# B&R Automation Studio project MIG1 (part 6)

```c
					ax = 0;
					for(k = 0 ; k < mgr->hrdw[i].AxisNum ; k++){

						if(mgr->pAxis[i]){
							if((mgr->pAxis[i][k].AxisID & 0x00FF)== SenderID){
								ax = &mgr->pAxis[i][k];
								break;

							}
						}

					}
					if(!ax)
						return 0;

#ifdef KK_SUPER_TRACE
					KK_Ind_RcvMsg_Cntr[i][k]++;
#endif
					/////////////////////////////////////////////////////////////
					// Parse message //
					// Firmware version
					if((*pRxCANidentifier) == 0xD80A0009){

						mgr->Firmware[i] = ((UDINT)pRxCANdata[1] + ((UDINT)pRxCANdata[0] <<16));
					}

					///////////////////////////////////////////////////////
					/*Received 32-bit variable*/
					else if((*pRxCANidentifier)& 0x800){ /* Check if 16 or 32-bit variable - bit 11 */

						if(pRxCANdata[0] == 0x090E){ /* Status Received */

							ax->Flag |= 0x0C; //bit 2 & 3  (* New Status received *)
							ax->DriveStatusRegisterL = pRxCANdata[1];
							ax->DriveStatusRegisterH = pRxCANdata[2];

						}
						else{ /* General variable received. Save address to Axis structure*/
							ax->Flag |= 0x01; //bit 0 (* New Variable received *)

							ax->VarAddress = pRxCANdata[0];
							ax->DataLow  = pRxCANdata[1];
							ax->DataHigh = pRxCANdata[2];

						}
					}
					////////////////////////////////////////////
					/*Received 16-bit variable*/
					else if(pRxCANdata[0] == 0x08FC){  /* MER register received */
						if(pRxCANdata[1] && 0xFFEF){ // Mask Serial comunnication error
							ax->Flag |= 0x02; //bit 1 (* New Error received *)
							ax->DriveErrorRegister = pRxCANdata[1];
						}
					}
					/***********/
					else if(pRxCANdata[0] == 0x0863){  /* PVT status register received*/

						ax->Flag |= 0x10; //bit 4 (* New PVT status received *)
						ax->PVTstatus = pRxCANdata[1];

					}
					/***********/
					else {  /* other variable received*/

						ax->Flag |= 0x01; //bit 0 (* New Variable received *)
						ax->VarAddress = pRxCANdata[0];
						ax->DataLow  = pRxCANdata[1];

					}

			}

		}
	}

return 1;
}

DINT ReadValue(char **p, DINT *val){

	if(*p == strchr(*p , 0x0D)){
		(*p)+= 2;
		return -1;
	}

	else {

		*val = 0;

		while( (**p != 0x0D) || (**p != 0x0A)){

			if((**p >= '0') && (**p <= '9')){
				*val = *val<<4;
				*val += (**p) - '0';
			}
			else if((**p >= 'A') && (**p <= 'F')){
				*val = *val<<4;
				*val += (**p) - 'A' + 10;
			}
			else{
				(*p)++;
				break;
			}

			(*p)++;

		}

	}

	(*p)++;

return 1;
}

DINT CalcUnits(TML_typ* tml){

	if( (tml->_cfg.rev_motor != 0.0) && (tml->_cfg.loopPeriod > 0)){
		tml->_int.kPos = (tml->_cfg.units * fabsf(tml->_cfg.rev_motor)) * tml->_cfg.rev_scale ;
		tml->_int.kVel = fabsf(tml->_int.kPos * tml->_cfg.loopPeriod);
		tml->_int.kAcc = tml->_int.kVel * tml->_cfg.loopPeriod ;
		//tml->_int.PVTPeriod = 0.02/ tml->_cfg.loopPeriod;
		tml->_int.PVTPeriod = (UINT)(tml->_cfg.PVTPeriod / tml->_cfg.loopPeriod + 0.5);
		return 1;
	}
	else
		return -1;

return 1;
}

DINT TML_InterpretMessage_UDP(TML_MGR_typ* mgr){

USINT *pCountRegister;
UDINT *pRxCANidentifier ;
UINT *pRxCANdata;
TML_Axis_typ *ax;
RS_Channel_typ *data , *data_sent;
USINT SenderID;
UINT i , k , n;
plcstring _str[128];
UINT adr ;
//UDINT val , *pVal;
USINT dataType; // 0 - no data , 1 - 16 data , 2 - 32 data
UINT *pUINT , val_UINT[2];

	if(!mgr)
		return -1;

	//pVal = &val;
	pUINT = &val_UINT[0];

	for(n = 0 ; n < 2 ; n++){ // Two channels

		data = ((RS_Channel_typ*)mgr->pRecData[n]) ;

		data_sent = ((RS_Channel_typ*)mgr->pSendData[n]) ;

		if(!data || !data_sent)
			continue;

		////////////////////////////////////////////////////////////////
		//////   New from 6 June 2023

		if(data->Len == 0)
			continue;

		mgr->hrdw[n].RXCount++;

		//if((data_sent->Len == 0)
		if(data->Len == 1){

			if(data->Data[0] == 0x4F){
				//&& (data_sent->Status == 0x1)){

				//LogTxt(&LogMgr, "ACK: F%d T%d" , (UDINT)mgr->hrdw[n].TXCountReadBack , (UDINT)mgr->hrdw[n].TXCount);
				data->Msg_ID ++;
				if(data_sent->Msg_ID == data->Msg_ID){

					mgr->hrdw[n].TXCountReadBack = mgr->hrdw[n].TXCount;
					data->Msg_ID = data_sent->Msg_ID;
					data->Status++;

				}else{

					mgr->hrdw[n].TXCountReadBack = mgr->hrdw[n].TXCount;
					data->Msg_ID = data_sent->Msg_ID;
					data_sent->Msg_Error++;
					data->Msg_Error++;
				}

			}
			else {
				data_sent->Trash_Cntr++;
				data->Trash_Cntr++;
			}

			data->Len = 0;
			continue;
		}

		//StreamToHex(data->Data, _str, data->Len);
		//LogTxt(&LogMgr, "%d-%d R: %s" , (UDINT) n , data->Len, _str);

		if(((data->Len != 10) && (data->Len != 12)&&(data->Len != 14) )){ // 16 or 32 bit TakeData only
			data->Trash_Cntr++;
			data->Len = 0;
			continue;

		}

		//if(!(data->Data[1] == 0x00 && data->Data[2] == 0xA1)){ // Not for me
		if(!((data->Data[1] == 0x00) && (data->Data[2] == (HOST_ID*0x10 +1)))){ // Not for me
			data->Trash_Cntr++;
			data->Len = 0;
			continue;
		}

		///////////////////////////////////////////////////////////////
		///////////////////////////////////////////////////////////////

		/*
		if((data_sent->Len == 0)
			&& (data->Len == 1)
			&& (data->Data[0] == 0x4F)){
			//&& (data_sent->Status == 0x1)){

			//LogTxt(&LogMgr, "ACK: F%d T%d" , (UDINT)mgr->hrdw[n].TXCountReadBack , (UDINT)mgr->hrdw[n].TXCount);

			mgr->hrdw[n].TXCountReadBack = mgr->hrdw[n].TXCount;

			data->Status++;

		}

		if(data->Len == 0)
			continue;

		//StreamToHex(data->Data, _str, data->Len);
		//LogTxt(&LogMgr, "%d-%d R: %s" , (UDINT) n , data->Len, _str);

		mgr->hrdw[n].RXCount++;

		if((data->Len == 1) // 0x4F - confirmation of cmd
			||((data->Len != 10) && (data->Len != 12)&&(data->Len != 14) )){ // 16 or 32 bit TakeData only

			data->Len = 0;
			return 0;

		}

		//if(!(data->Data[1] == 0x00 && data->Data[2] == 0xA1)){ // Not for me
		if(!((data->Data[1] == 0x00) && (data->Data[2] == (HOST_ID*0x10 +1)))){ // Not for me
			data->Len = 0;
			return;
		}

		*/
		///////////////// to dziala ///////////////////////
		dataType = 0;
		//val = 0;
		val_UINT[0] = 0;
		val_UINT[1] = 0;
		switch(data->Data[3]){

			case 0xB4: // TakeData 16 bit 0r 32 bit

				SenderID = (UINT)data->Data[6] + (UINT)data->Data[5] * 0x100;
				SenderID /= 0x10;

				adr = (UINT)data->Data[8] + (UINT)data->Data[7] * 0x100;

				switch(data->Data[4]){

					case 0x04: // 16 bit data

						*((char*)pUINT) = data->Data[10];
						*((char*)pUINT + 1) = data->Data[9];

						dataType = 1;

					break;

					case 0x05: // 32 bit data

						//val = (UINT)data->Data[10] + (UINT)data->Data[9] * 0x100 \
							//+ (UINT)data->Data[12] * 0x10000  + (UINT)data->Data[11] * 0x1000000;

						//*((char*)pVal) = data->Data[10];
						//*((char*)pVal + 1) = data->Data[9];
						//*((char*)pVal + 2) = data->Data[12];
						//*((char*)pVal + 3) = data->Data[11];

						*((char*)pUINT) = data->Data[10];
						*((char*)pUINT + 1) = data->Data[9];
						*((char*)pUINT + 2) = data->Data[12];
						*((char*)pUINT + 3) = data->Data[11];

						dataType = 2;

					break;

					default:

					break;
				}

				//LogTxt(&LogMgr, "D1:%d A:%X U: %X , %X" , (DINT)SenderID , (UINT)adr , val_UINT[0] , val_UINT[1]);

			break;

			case 0xD4: // TakeData2 16 bit
			case 0xD5: // TakeData2 32 bit

				SenderID = data->Data[4];

				adr = (UINT)data->Data[6] + (UINT)data->Data[5] * 0x100;

				switch(data->Data[3]){

					case 0xD4: // TakeData2 16 bit

						*((char*)pUINT) = data->Data[8];
						*((char*)pUINT + 1) = data->Data[7];

						dataType = 1;

					break;

					case 0xD5: // TakeData2 32 bit

						*((char*)pUINT) = data->Data[8];
						*((char*)pUINT + 1) = data->Data[7];
						*((char*)pUINT + 2) = data->Data[10];
						*((char*)pUINT + 3) = data->Data[9];

						dataType = 2;

					break;

				}

				//LogTxt(&LogMgr, "D2:%d A:%X U: %X , %X" , (DINT)SenderID , (UINT)adr  , val_UINT[0] , val_UINT[1]);

			break;

		}

		data->Len = 0;

		///////////////////////////////////////////////////////////////////////////
		ax = 0;
		for(k = 0 ; k < mgr->hrdw[n].AxisNum ; k++){

			if(mgr->pAxis[n]){
				if((mgr->pAxis[n][k].AxisID & 0x00FF)== SenderID){
					ax = &mgr->pAxis[n][k];
					//LogTxt(&LogMgr, "Axis Chan: %d Item: %d Node:%d Type: %d" , (UDINT) n , (UDINT)k , (UDINT)SenderID , (UDINT)dataType);
					break;

				}
			}

		}

		if(!ax)
			return 0;

		//ax->VarAddress = dataType;
		//ax->PVTstatus = SenderID;
		//return;

		//LogTxt(&LogMgr, "Type: %d Adr: %X U1:%X U2: %X " ,(UDINT)dataType , (UDINT)adr , (UDINT)val_UINT[0] , (UDINT)val_UINT[1] );

		switch(dataType){

			case 0: // nothing

			break;

			case 1: // 16 bit

				if(adr == 0x08FC){  /* MER register received */

					ax->AxisState = val_UINT[0] & 0xA000 ; // only enable and undervoltage

					if(val_UINT[0] & 0xFFEF){ // Mask Serial comunnication error
					//if(val_UINT[0] & 0x5FEF){ // Mask Serial comunnication error and  enable and undervoltage
						ax->Flag |= 0x02; //bit 1 (* New Error received *)
						ax->DriveErrorRegister = val_UINT[0];
					}
				}
				/***********/
				else if(adr == 0x0863){  /* PVT status register received*/

					ax->Flag |= 0x10; //bit 4 (* New PVT status received *)
					ax->PVTstatus = val_UINT[0];

				}
				/***********/
				else {	/* other variable received*/

					ax->Flag |= 0x01; //bit 0 (* New Variable received *)
					ax->VarAddress = adr;
					ax->DataLow  = val_UINT[0];

				}
			break;

			case 2: // 32 bit

				if(adr == 0x090E){ // Status Received

					ax->Flag |= 0x0C; //bit 2 & 3  New Status received
					ax->DriveStatusRegisterL = val_UINT[0];
					ax->DriveStatusRegisterH = val_UINT[1];

				}
				else{ // General variable received. Save address to Axis structure
					ax->Flag |= 0x01; //bit 0  New Variable received

					ax->VarAddress = adr;
					ax->DataLow  = val_UINT[0];
					ax->DataHigh = val_UINT[1];

				}

			break;

		}

		///////////////////////////////

	}

return 1;

}

DINT TML_BuildMessage_UDP(UINT AxisID, UINT Channel , UINT OpCode, UINT Address, UDINT OpData1, UDINT OpData2, USINT MessageLength, USINT DataType, TML_MGR_typ* mgr ){
UINT i;
RS_Channel_typ* data;
plcstring _str[128];

	if(!mgr)
		return -1;

	if(Channel > 1)
		return -2;

	if(!mgr->pSendData)
		return -3;

	////  Super Trace
#ifdef KK_SUPER_TRACE

	if(OpCode == 0x0402)
		LogTxt(&LogMgr , "Axis %d Reset" , (UDINT)AxisID);

	else if(OpCode == TML_set_Param_0_int+7)
		LogTxt(&LogMgr , "Axis %d Set Tmr %d" , (UDINT)AxisID , OpData1);

	if((OpCode == 0x0410) || (OpCode == 0x0510))
			KK_StrangeCode_Cntr++;

	KK_BuiltMsg_Cntr++;

	if((AxisID < 32) && (Channel < 2))
		KK_Ind_BuiltMsg_Cntr[Channel][AxisID]++;

#endif

		data = ((RS_Channel_typ*)mgr->pSendData[Channel]) ;

		if(!data)
			return -3;

		if(data->Len != 0){
			data->Trash_Cntr ++;
			return  0;
		}

		//data->Len = 0;

		AxisID = AxisID * 0x10;
		data->Data[2] = (char)*((USINT*)&AxisID);
		data->Data[1] = (char)*((USINT*)&AxisID + 1);

		data->Data[4] = (char)*((USINT*)&OpCode);
		data->Data[3] = (char)*((USINT*)&OpCode + 1);

		if((OpCode == 0xB004) // GiveMeData = 16 bit TML data
			|| (OpCode == 0xB005)){ // GiveMeData = 32 bit TML data

			DataType = 2;
			OpData1 = Address * 0x10000 + (HOST_ID * 0x10) + 1; //0x03B7 - variable adress , 10 - Host Address , 1 - Host

		}

		switch (DataType){

			case 1:/* Send 16-bit data*/

				//LogTxt(&LogMgr, "MT1:%d OP:%X V:%d" , (DINT)AxisID , (UDINT)OpCode , (UDINT)OpData1);

				data->Data[0] = 0x06;

				data->Data[6] = (char)*((USINT*)&OpData1);
				data->Data[5] = (char)*((USINT*)&OpData1 + 1);

				data->Data[7] = 0;
				for(i = 0; i <= data->Data[0] ; i++)
					data->Data[7] += data->Data[i];

			break;

			case 2:/* Send 32-bit data*/

				//LogTxt(&LogMgr, "MT2:%d OP:%X V:%d" , (DINT)AxisID , (UINT)Address , (UDINT)OpCode ,(UDINT)OpData1);

				data->Data[0] = 0x08;

				data->Data[6] = (char)*((USINT*)&OpData1);
				data->Data[5] = (char)*((USINT*)&OpData1 + 1);
				data->Data[8] = (char)*((USINT*)&OpData1 + 2);
				data->Data[7] = (char)*((USINT*)&OpData1 + 3);

				data->Data[9] = 0;
				for(i = 0; i <= data->Data[0] ; i++)
					data->Data[9] += data->Data[i];

			break;

			default: // just command

				data->Data[0] = 0x04;

				data->Data[5] = 0;
				for(i = 0; i <= data->Data[0] ; i++)
					data->Data[5] += data->Data[i];

			break;

		}

		data->Len = data->Data[0]+2;

		//StreamToHex(data->Data, _str, data->Data[0]+2);
		//LogTxt(&LogMgr, "S: %s" , _str);

		if(OpCode != 0x0402) // not RESET command
			mgr->hrdw[Channel].TXCount ++; //= mgr->hrdw[Channel].TXCountReadBack+1;

		data->Msg_ID++;

	return 1;

}
```

### Program Logical/TML_Cfg (ANSIC)

#### TML_Cfg.c - Init, cyclic, exit code
```c
#include <bur/plctypes.h>

#ifdef _DEFAULT_INCLUDES
	#include <AsDefault.h>
#endif

#include <..\GlobalDef.h>
#include <..\GlobalDecl.h>

#include <..\Lib\Statelib.c>
#include <..\Lib\LoggerLib.c>
#include <..\Lib\WSI_lib.c>
//#include <..\Lib\utilityLib\bgdebug.h>

// Only For ESTOP from Universla Controller
_GLOBAL plcbit ESTOP_out;

void AssignMtrErrorText(char* txt , UDINT i , UDINT val );

_LOCAL plcbit KK_ClearErrors;

////    Super Mini Head
void _INIT ProgramInit(void)
{int i;

	//hardware.Inputs[5] = 1; //ControlModule_Estop_Active
	//hardware.Outputs[7];  // Estop Output

	ESTOP_out = 1;

	TML_mgr[0].pLog = TML_mgr[0].pLog;
	VectorStateMach[0].fParam[0] = VectorStateMach[0].fParam[0];
	TML_MTR_INST[0].AnInp[0] = TML_MTR_INST[0].AnInp[0] ;
	AxisCh[0].AxisID = 0;
	LogMgr.Cmd.Refresh = LogMgr.Cmd.Refresh;

	/***********************************************************/
	//LogTxt(&LogMgr , "Start TML Cfg %d " , 1);
	LoggerInit(&LogMgr, &LogID, "LogBook1", 2000);
	///////////////////////////////////////
	/***********************************************************/

	/////////////////////////////////

	i = TML_AX_OSC; // UnvCntrl_SMH_19-10_25.m.zip

	strcpy(TML_MTR_INST[i].Name , "OSC");

	// Analog Feedback from REF
	TML_MTR_INST[i]._cfg.loopPeriod = 0.001;

	TML_MTR_INST[i]._cfg.units = 1024 * 4;

	//TML_MTR_INST[i]._cfg.rev_motor = -62.0;
	//TML_MTR_INST[i]._cfg.rev_scale = -1.0/ (0.5 * 25.4) ;

	TML_MTR_INST[i]._cfg.rev_motor = 1.0;
	TML_MTR_INST[i]._cfg.rev_scale = 1.0/ (100.0) ;

	TML_MTR_INST[i]._cfg.maxVel = 6000.0/60.0    /TML_MTR_INST[i]._cfg.rev_motor/ TML_MTR_INST[i]._cfg.rev_scale;

	// (tml->_cfg.units * fabsf(tml->_cfg.rev_motor) * tml->_cfg.rev_scale   * tml->_cfg.loopPeriod * V = 60000/60.0 * TML_MTR_INST[i]._cfg.loopPeriod * 	TML_MTR_INST[i]._cfg.units ;

	TML_MTR_INST[i]._cfg.maxAcc = TML_MTR_INST[i]._cfg.maxVel * 100.0 ;
	TML_MTR_INST[i]._cfg.absLastPos = OLD_MTR_POS[i];
	//TML_MTR_INST[i]._cfg.absFbk = 2; // absolute
	TML_MTR_INST[i]._cfg.absFbk = 0;

	TML_MTR_INST[i]._cfg.HeartBeat = 0.4;
	TML_MTR_INST[i]._cfg.PVTPeriod = 0.08;

	strcpy(TML_MTR_INST[i]._cfg.programName , "1521_SMH_OSC.sw");
	//TML_MTR_INST[i].ProgramVersion = ASC2UDINT("1521");
	TML_MTR_INST[i].ProgramVersion = ASC2UDINT("1525");

	TML_MTR_INST[i]._cfg.Appl_ID_adr = 0x7FCF;

	//TML_MTR_INST[i].FirmwareVersion = ASC2UDINT("674C");  //0x674B
	TML_MTR_INST[i].FirmwareVersion = ASC2UDINT("6A2B");  //0x674B
	TML_MTR_INST[i]._cfg.NotAutoDownload = 1;

	/*
	strcpy(TML_MTR_INST[i].Name , "OSC");

	// Analog Feedback from REF
	TML_MTR_INST[i]._cfg.loopPeriod = 0.001;

	TML_MTR_INST[i]._cfg.units = 1024 * 4;

	//This is from BPV
	TML_MTR_INST[i]._cfg.rev_motor = (-75.0/19.0) * 50.0;
	//TML_MTR_INST[i]._cfg.rev_scale = -1.0/ (0.625 * 25.4 *M_PI) ; // To jest dobrze
	TML_MTR_INST[i]._cfg.rev_scale = 1.0/ (0.625 * 25.4 *M_PI) ; // A to tylko do eksperymentu

	TML_MTR_INST[i]._cfg.maxVel = 8000.0/60.0/TML_MTR_INST[i]._cfg.rev_motor/ TML_MTR_INST[i]._cfg.rev_scale;
	TML_MTR_INST[i]._cfg.maxAcc = TML_MTR_INST[i]._cfg.maxVel * 10.0 ;
	TML_MTR_INST[i]._cfg.absLastPos = OLD_MTR_POS[TML_AX_OSC];
	TML_MTR_INST[i]._cfg.pAbsLastPos = &OLD_MTR_POS[i];

	TML_MTR_INST[i]._int.kVolt = 1365.0;

	TML_MTR_INST[i]._cfg.absFbk = 10;

	TML_MTR_INST[i]._cfg.HeartBeat = 0.4;
	//TML_MTR_INST[i]._cfg.PVTPeriod = 0.08;

	strcpy(TML_MTR_INST[i]._cfg.programName , "1821_BPV2_OSC.sw");
	TML_MTR_INST[i].ProgramVersion = ASC2UDINT("1821");

	TML_MTR_INST[i].FirmwareVersion = ASC2UDINT("674C");  //0x674B
	TML_MTR_INST[i]._cfg.NotAutoDownload = 1;
	*/

	////////////////////////////////////////
	i = TML_AX_TVL; // /// UnvCntrl_SMH_19-10_25.m.zip

	strcpy(TML_MTR_INST[i].Name , "TVL");
	// Back EMF
	TML_MTR_INST[i]._cfg.loopPeriod = 0.0005; // Slow loop
	TML_MTR_INST[i]._cfg.units = 1024 * 4; //
	TML_MTR_INST[i]._cfg.rev_motor = -231.0;
	TML_MTR_INST[i]._cfg.rev_scale = (36.0/33.0) /( 1.25 * 25.4 * M_PI) ;

	TML_MTR_INST[i]._cfg.maxVel = fabsf(4500.0/60.0/TML_MTR_INST[i]._cfg.rev_motor/ TML_MTR_INST[i]._cfg.rev_scale);
	TML_MTR_INST[i]._cfg.maxAcc = TML_MTR_INST[i]._cfg.maxVel * 10.0 ;
	TML_MTR_INST[i]._cfg.absLastPos = OLD_MTR_POS[i];
	TML_MTR_INST[i]._cfg.absFbk = 2;

	//TML_MTR_INST[i]._cfg.HeartBeat = 0.08;
	TML_MTR_INST[i]._cfg.HeartBeat = 0.5;

	strcpy(TML_MTR_INST[i]._cfg.programName , "1525_SMH_TVL.sw");
	TML_MTR_INST[i].ProgramVersion = ASC2UDINT("1525");

	TML_MTR_INST[i].FirmwareVersion = ASC2UDINT("6A2B");  //0x674B
	TML_MTR_INST[i]._cfg.Appl_ID_adr = 0x7FCF;
	TML_MTR_INST[i]._cfg.NotAutoDownload = 1;

	/*
	strcpy(TML_MTR_INST[i].Name , "TVL");

	// Corrected 29May19
	//TML_MTR_INST[i]._cfg.loopPeriod = 0.0005; // Slow loop
	TML_MTR_INST[i]._cfg.loopPeriod = 0.001; // Slow loop
	// It was in BPV
	TML_MTR_INST[i]._cfg.units = 1024 * 4; //
	TML_MTR_INST[i]._cfg.rev_motor = 156;
	TML_MTR_INST[i]._cfg.rev_scale = 1.0 /( 1.25 * 25.4 * M_PI) ;

	TML_MTR_INST[i]._cfg.maxVel = fabsf(4500.0/60.0/TML_MTR_INST[i]._cfg.rev_motor/ TML_MTR_INST[i]._cfg.rev_scale);
	TML_MTR_INST[i]._cfg.maxAcc = TML_MTR_INST[i]._cfg.maxVel * 10.0 ;
	TML_MTR_INST[i]._cfg.absLastPos = OLD_MTR_POS[i];
	TML_MTR_INST[i]._cfg.absFbk = 2;

	TML_MTR_INST[i]._cfg.HeartBeat = 0.2;

	strcpy(TML_MTR_INST[i]._cfg.programName , "1625_BPV2_TVL.sw");
	TML_MTR_INST[i].ProgramVersion = ASC2UDINT("1625");

	TML_MTR_INST[i].FirmwareVersion = ASC2UDINT("6A2B");  //0x674B
	TML_MTR_INST[i]._cfg.Appl_ID_adr = 0x7FCF;
	TML_MTR_INST[i]._cfg.NotAutoDownload = 1;
	/////////////////////////////////////////////////////////////
	*/

	///////////////////////////////////////////////////
	i = TML_AX_INDX; // UnvCntrl_SMH_19-10_25.m.zip

	strcpy(TML_MTR_INST[i].Name , "INDX");

	// Analog Feedback from REF
	TML_MTR_INST[i]._cfg.loopPeriod = 0.001;

	TML_MTR_INST[i]._cfg.units = 1024 * 4;
	TML_MTR_INST[i]._cfg.rev_motor = 3.9 * 50 ;
	TML_MTR_INST[i]._cfg.rev_scale = -1.0/ (0.625 * 25.4 *M_PI) ;
	TML_MTR_INST[i]._cfg.maxVel = fabsf(8000.0/60.0/TML_MTR_INST[i]._cfg.rev_motor/ TML_MTR_INST[i]._cfg.rev_scale);
	TML_MTR_INST[i]._cfg.maxAcc = TML_MTR_INST[i]._cfg.maxVel * 10.0 ;
	TML_MTR_INST[i]._cfg.absLastPos = OLD_MTR_POS[i];
	TML_MTR_INST[i]._cfg.absFbk = 2;

	TML_MTR_INST[i]._cfg.HeartBeat = 0.5;
	TML_MTR_INST[i]._cfg.PVTPeriod = 0.08;

	strcpy(TML_MTR_INST[i]._cfg.programName , "1523_SMH_WRST.sw");
	TML_MTR_INST[i].ProgramVersion = ASC2UDINT("1523");

	TML_MTR_INST[i].FirmwareVersion = ASC2UDINT("674C");  //0x674B
	TML_MTR_INST[i]._cfg.NotAutoDownload = 1;

	///////////
	TML_MTR_INST[i].ProgramVersion = ASC2UDINT("1525");

	TML_MTR_INST[i]._cfg.Appl_ID_adr = 0x7FCF;

	//TML_MTR_INST[i].FirmwareVersion = ASC2UDINT("674C");  //0x674B
	TML_MTR_INST[i].FirmwareVersion = ASC2UDINT("6A2B");  //0x674B
	TML_MTR_INST[i]._cfg.NotAutoDownload = 1;

	/*

	// Analog Feedback from REF
	TML_MTR_INST[i]._cfg.loopPeriod = 0.001;

	TML_MTR_INST[i]._cfg.units = 500 * 4;
	TML_MTR_INST[i]._cfg.rev_motor = 24;
	TML_MTR_INST[i]._cfg.rev_scale = 1.0/5.0;
	TML_MTR_INST[i]._cfg.maxVel = 10000.0; //
	TML_MTR_INST[i]._cfg.maxAcc = 100.0;
	TML_MTR_INST[i]._cfg.absFbk = 0;

	TML_MTR_INST[i]._cfg.HeartBeat = 0.4;

	strcpy(TML_MTR_INST[i]._cfg.programName , "0326_BPV_WP.sw");
	TML_MTR_INST[i].ProgramVersion = ASC2UDINT("0326");

	TML_MTR_INST[i].FirmwareVersion = ASC2UDINT("6A2B");
	TML_MTR_INST[i]._cfg.Appl_ID_adr = 0x7FCF;
	TML_MTR_INST[i]._cfg.NotAutoDownload = 1;
	*/
	////////////////////////////////////////////
	i = TML_AX_AHC; // UnvCntrl_SMH_19-10_25.m.zip

	strcpy(TML_MTR_INST[i].Name , "AHC");

	// Analog Feedback from REF
	TML_MTR_INST[i]._cfg.loopPeriod = 0.001;
	TML_MTR_INST[i]._cfg.units = 4096;
	TML_MTR_INST[i]._cfg.rev_motor = 1;
	TML_MTR_INST[i]._cfg.rev_scale = 1.0/5.0;
	TML_MTR_INST[i]._cfg.maxVel = 1500.0;
	TML_MTR_INST[i]._cfg.maxAcc = TML_MTR_INST[i]._cfg.maxVel * 10.0;
	//TML_MTR_INST[i]._cfg.satpMax = 27853; // KPP bylo Stauration of proportional gain
	TML_MTR_INST[i]._cfg.satpMax = 32000; // KPP bylo Stauration of proportional gain
	//TML_MTR_INST[i]._cfg.kppMax = 32000; // KPP bylo Stauration of proportional gain
	//TML_MTR_INST[i]._cfg.kipMax = 200; // KPP bylo Stauration of proportional gain
	TML_MTR_INST[i]._cfg.kppMax = 32000;
	TML_MTR_INST[i]._cfg.kipMax = 1000;
	TML_MTR_INST[i]._cfg.absFbk = 0;

	TML_MTR_INST[i]._cfg.HeartBeat = 0.8;

	//TML_MTR_INST[i]._cfg.signFilter = curCfg->Param[parAVC_FbkFilter].val[0];

	//U_BEND_HP_PINS
	strcpy(TML_MTR_INST[i]._cfg.programName , "1526_SMH_AVC.sw");
	TML_MTR_INST[i].ProgramVersion = ASC2UDINT("1526");

	TML_MTR_INST[i].FirmwareVersion = ASC2UDINT("6A2B");  //0x674C , 514D
	TML_MTR_INST[i]._cfg.Appl_ID_adr = 0x7FCF;
	TML_MTR_INST[i]._cfg.NotAutoDownload = 1;

	///////////
	TML_MTR_INST[i].ProgramVersion = ASC2UDINT("1525");

	TML_MTR_INST[i]._cfg.Appl_ID_adr = 0x7FCF;

	//TML_MTR_INST[i].FirmwareVersion = ASC2UDINT("674C");  //0x674B
	TML_MTR_INST[i].FirmwareVersion = ASC2UDINT("6A2B");  //0x674B
	TML_MTR_INST[i]._cfg.NotAutoDownload = 1;
	///////////////////

	//TML_MTR_INST[i]._cfg.sftLimitPos = 0.0;
	//TML_MTR_INST[i]._cfg.sftLimitNeg = 0.0;

	//TML_MTR_INST[i]._cfg.AnalLimitPos = 3900;
	//TML_MTR_INST[i]._cfg.AnalLimitNeg = 100;

	TML_MTR_INST[i]._cfg.MtrType = 1 ; // 3phase brusshless

	/////

	TML_MTR_INST[i]._cfg.loopPeriod = 0.0005; // Slow loop
	TML_MTR_INST[i]._cfg.units = 1024 * 4; //
	TML_MTR_INST[i]._cfg.rev_motor = -231.0;
	TML_MTR_INST[i]._cfg.rev_scale = (36.0/33.0) /( 1.25 * 25.4 * M_PI) ;

	TML_MTR_INST[i]._cfg.maxVel = fabsf(4500.0/60.0/TML_MTR_INST[i]._cfg.rev_motor/ TML_MTR_INST[i]._cfg.rev_scale);
	TML_MTR_INST[i]._cfg.maxAcc = TML_MTR_INST[i]._cfg.maxVel * 10.0 ;
	TML_MTR_INST[i]._cfg.absLastPos = OLD_MTR_POS[i];
	TML_MTR_INST[i]._cfg.absFbk = 2;

	//TML_MTR_INST[i]._cfg.HeartBeat = 0.08;
	TML_MTR_INST[i]._cfg.HeartBeat = 0.5;

	strcpy(TML_MTR_INST[i]._cfg.programName , "1525_SMH_TVL.sw");
	TML_MTR_INST[i].ProgramVersion = ASC2UDINT("1525");

	TML_MTR_INST[i].FirmwareVersion = ASC2UDINT("6A2B");  //0x674B
	TML_MTR_INST[i]._cfg.Appl_ID_adr = 0x7FCF;
	TML_MTR_INST[i]._cfg.NotAutoDownload = 1;

	/*
	// Analog Feedback from REF
	TML_MTR_INST[i]._cfg.loopPeriod = 0.001;
	TML_MTR_INST[i]._cfg.units = 4096;
	TML_MTR_INST[i]._cfg.rev_motor = 1;
	TML_MTR_INST[i]._cfg.rev_scale = 1.0/5.0;
	TML_MTR_INST[i]._cfg.maxVel = 1500.0;
	TML_MTR_INST[i]._cfg.maxAcc = TML_MTR_INST[i]._cfg.maxVel * 10.0;
	//TML_MTR_INST[i]._cfg.satpMax = 27853; // KPP bylo Stauration of proportional gain
	TML_MTR_INST[i]._cfg.satpMax = 32000; // KPP bylo Stauration of proportional gain
	//TML_MTR_INST[i]._cfg.kppMax = 32000; // KPP bylo Stauration of proportional gain
	//TML_MTR_INST[i]._cfg.kipMax = 200; // KPP bylo Stauration of proportional gain
	TML_MTR_INST[i]._cfg.kppMax = 32000;
	TML_MTR_INST[i]._cfg.kipMax = 1000;
	TML_MTR_INST[i]._cfg.absFbk = 0;

	TML_MTR_INST[i]._cfg.HeartBeat = 0.8;

	//TML_MTR_INST[i]._cfg.signFilter = curCfg->Param[parAVC_FbkFilter].val[0];

	strcpy(TML_MTR_INST[i]._cfg.programName , "1526_SMH_AVC.sw");
	TML_MTR_INST[i].ProgramVersion = ASC2UDINT("1526");

	TML_MTR_INST[i].FirmwareVersion = ASC2UDINT("6A2B");  //0x674C , 514D
	TML_MTR_INST[i]._cfg.Appl_ID_adr = 0x7FCF;
	TML_MTR_INST[i]._cfg.NotAutoDownload = 1;

	//TML_MTR_INST[i]._cfg.sftLimitPos = 0.0;
	//TML_MTR_INST[i]._cfg.sftLimitNeg = 0.0;

	TML_MTR_INST[i]._cfg.AnalLimitPos = 3900;
	TML_MTR_INST[i]._cfg.AnalLimitNeg = 100;

	TML_MTR_INST[i]._cfg.MtrType = 1 ; // 3phase brusshless
	*/

	////////////////////////////////////////////
	i = TML_AX_WF; // UnvCntrl_SMH_19-10_25.m.zip

	strcpy(TML_MTR_INST[i].Name , "WF");

	// Analog Feedback from REF
	TML_MTR_INST[i]._cfg.loopPeriod = 0.001;
	TML_MTR_INST[i]._cfg.units = 1024 * 4; //
	//TML_MTR_INST[i]._cfg.rev_motor = 35;

	TML_MTR_INST[i]._cfg.maxVel = 400 * 25.4/ 60.0; //// 520 ipm
	TML_MTR_INST[i]._cfg.maxAcc = TML_MTR_INST[i]._cfg.maxVel * 10.0;
	TML_MTR_INST[i]._cfg.absFbk = 0;

	TML_MTR_INST[i]._cfg.HeartBeat = 0.4;

	strcpy(TML_MTR_INST[i]._cfg.programName , "1522_SMH_WF.sw");
	TML_MTR_INST[i].ProgramVersion = ASC2UDINT("1522");

	TML_MTR_INST[i].FirmwareVersion = ASC2UDINT("674C");
	TML_MTR_INST[i]._cfg.Appl_ID_adr = 0x7FCF;
	TML_MTR_INST[i]._cfg.NotAutoDownload = 1;

	////

	TML_MTR_INST[i]._cfg.loopPeriod = 0.0005; // Slow loop
	TML_MTR_INST[i]._cfg.units = 1024 * 4; //
	TML_MTR_INST[i]._cfg.rev_motor = -231.0;
	TML_MTR_INST[i]._cfg.rev_scale = (36.0/33.0) /( 1.25 * 25.4 * M_PI) ;

	TML_MTR_INST[i]._cfg.maxVel = fabsf(4500.0/60.0/TML_MTR_INST[i]._cfg.rev_motor/ TML_MTR_INST[i]._cfg.rev_scale);
	TML_MTR_INST[i]._cfg.maxAcc = TML_MTR_INST[i]._cfg.maxVel * 10.0 ;
	TML_MTR_INST[i]._cfg.absLastPos = OLD_MTR_POS[i];
	TML_MTR_INST[i]._cfg.absFbk = 2;

	//TML_MTR_INST[i]._cfg.HeartBeat = 0.08;
	TML_MTR_INST[i]._cfg.HeartBeat = 0.5;

	strcpy(TML_MTR_INST[i]._cfg.programName , "1525_SMH_TVL.sw");
	TML_MTR_INST[i].ProgramVersion = ASC2UDINT("1525");

	TML_MTR_INST[i].FirmwareVersion = ASC2UDINT("6A2B");  //0x674B
	TML_MTR_INST[i]._cfg.Appl_ID_adr = 0x7FCF;
	TML_MTR_INST[i]._cfg.NotAutoDownload = 1;

	/*
	// Analog Feedback from REF
	TML_MTR_INST[i]._cfg.loopPeriod = 0.001;
	TML_MTR_INST[i]._cfg.units = 1024 * 4; //

	TML_MTR_INST[i]._cfg.rev_scale = 1.0 /( 0.75 * 25.4 * M_PI) ;
	TML_MTR_INST[i]._cfg.rev_motor = 35.0;

	TML_MTR_INST[i]._cfg.maxVel = 520 * 25.4/ 60.0; //// 520 ipm
	TML_MTR_INST[i]._cfg.maxAcc = TML_MTR_INST[i]._cfg.maxVel * 4.0;
	TML_MTR_INST[i]._cfg.absFbk = 0;

	TML_MTR_INST[i]._cfg.HeartBeat = 0.4;

	strcpy(TML_MTR_INST[i]._cfg.programName , "0325_BPV_WF.sw");
	TML_MTR_INST[i].ProgramVersion = ASC2UDINT("0325");

	TML_MTR_INST[i].FirmwareVersion = ASC2UDINT("6A2B");
	TML_MTR_INST[i]._cfg.Appl_ID_adr = 0x7FCF;
	TML_MTR_INST[i]._cfg.NotAutoDownload = 1;
	*/
	/***********************************************************/
	/***************************************************************/
	/////////////////////////////////////////////////////////////////

	TML_MTR_INST[TML_AX_TVL].pState = &VectorStateMach[VECT_AX_TVL];
	TML_MTR_INST[TML_AX_OSC].pState = &VectorStateMach[VECT_AX_OSC];
	TML_MTR_INST[TML_AX_INDX].pState = &VectorStateMach[VECT_AX_INDX];
	TML_MTR_INST[TML_AX_AHC].pState = &VectorStateMach[VECT_AX_AHC];
	TML_MTR_INST[TML_AX_WF].pState = &VectorStateMach[VECT_AX_WF];

	for(i=0 ; i < VECTORS_NUM; i++)
		VectorStateMach[i].Indx = i;

	strcpy(VectorStateMach[VECT_AX_TVL].Name , TML_MTR_INST[TML_AX_TVL].Name);
	strcpy(VectorStateMach[VECT_AX_OSC].Name , TML_MTR_INST[TML_AX_OSC].Name);
	strcpy(VectorStateMach[VECT_AX_INDX].Name , TML_MTR_INST[TML_AX_INDX].Name);
	strcpy(VectorStateMach[VECT_AX_AHC].Name , TML_MTR_INST[TML_AX_AHC].Name);
	strcpy(VectorStateMach[VECT_AX_WF].Name , TML_MTR_INST[TML_AX_WF].Name);

	TML_mgr[0].hrdw[0].AxisNum = 0;
	TML_mgr[0].hrdw[1].AxisNum = 5;

	TML_mgr[0].pAxis[0] = 0;
	TML_mgr[0].pAxis[1] = &AxisCh[0];

	TML_mgr[0].pTML[0] = 0;
	TML_mgr[0].pTML[1] = &TML_MTR_INST[0];

	//AxisCh[TML_AX_TVL].AxisID	= 25;	// BPV2 - TVL
	AxisCh[TML_AX_TVL].AxisID	= 17;	// tylko w biurze
	AxisCh[TML_AX_OSC].AxisID 	= 14;	// BPV2 - OSC
	//AxisCh[TML_AX_OSC].AxisID 	= 21;	// BPV2 - OSC
	AxisCh[TML_AX_INDX].AxisID 	= 12;	// BPV2 - WP
	//AxisCh[TML_AX_INDX].AxisID 	= 6;	// BPV2 - WP
	AxisCh[TML_AX_AHC].AxisID 	= 16; 	// BPV2 - AVC
	AxisCh[TML_AX_WF].AxisID 	= 15;	// BPV2 - WF
	//AxisCh[TML_AX_WF].AxisID 	= 5;	// BPV2 - WF

	//////////////////////////////////////////////////////

	TML_MTR_INST[TML_AX_TVL].Disable = 0;
	TML_MTR_INST[TML_AX_OSC].Disable = 0;
	TML_MTR_INST[TML_AX_INDX].Disable = 0;
	TML_MTR_INST[TML_AX_AHC].Disable = 0;
	TML_MTR_INST[TML_AX_WF].Disable = 0;

	VectorStateMach[VECT_AX_TVL].simul = 0;
	VectorStateMach[VECT_AX_OSC].simul = 0;
	VectorStateMach[VECT_AX_INDX].simul = 0;
	VectorStateMach[VECT_AX_AHC].simul = 0;
	VectorStateMach[VECT_AX_WF].simul = 0;

	VectorStateMach[VECT_AX_TVL].testMode = 0;
	VectorStateMach[VECT_AX_OSC].testMode = 0;
	VectorStateMach[VECT_AX_INDX].testMode = 0;
	VectorStateMach[VECT_AX_AHC].testMode = 0;
	VectorStateMach[VECT_AX_WF].testMode = 0;

	///////////////////////////////////////////////////////////
	/// Tak jest w BPV2

	/*
	AxisCh[TML_AX_TVL].AxisID	= 25;
	AxisCh[TML_AX_OSC].AxisID 	= 21;
	AxisCh[TML_AX_AVC].AxisID 	= 26;
	AxisCh[TML_AX_WRST].AxisID 	= 23;

	AxisCh[TML_AX_INDX].AxisID 	= 22;
	AxisCh[TML_AX_INDX_1].AxisID 	= 24;

	AxisCh[TML_AX_WF].AxisID 	= 5;
	AxisCh[TML_AX_WP].AxisID 	= 6;
	AxisCh[TML_AX_WF_1].AxisID 	= 7;
	AxisCh[TML_AX_WP_1].AxisID 	= 8;
	*/

}

#if 0
void _INIT ProgramInit(void)
{int i;

	//hardware.Inputs[5] = 1; //ControlModule_Estop_Active
	//hardware.Outputs[7];  // Estop Output

	ESTOP_out = 1;

	TML_mgr[0].pLog = TML_mgr[0].pLog;
	VectorStateMach[0].fParam[0] = VectorStateMach[0].fParam[0];
	TML_MTR_INST[0].AnInp[0] = TML_MTR_INST[0].AnInp[0] ;
	AxisCh[0].AxisID = 0;
	LogMgr.Cmd.Refresh = LogMgr.Cmd.Refresh;

	/***********************************************************/
	//LogTxt(&LogMgr , "Start TML Cfg %d " , 1);
	LoggerInit(&LogMgr, &LogID, "LogBook1", 2000);
	///////////////////////////////////////
	/***********************************************************/

	/////////////////////////////////

	i = TML_AX_OSC;

	strcpy(TML_MTR_INST[i].Name , "OSC");

	// Analog Feedback from REF
	TML_MTR_INST[i]._cfg.loopPeriod = 0.001;

	TML_MTR_INST[i]._cfg.units = 1024 * 4;

	//This is from BPV
	TML_MTR_INST[i]._cfg.rev_motor = (-75.0/19.0) * 50.0;
	//TML_MTR_INST[i]._cfg.rev_scale = -1.0/ (0.625 * 25.4 *M_PI) ; // To jest dobrze
	TML_MTR_INST[i]._cfg.rev_scale = 1.0/ (0.625 * 25.4 *M_PI) ; // A to tylko do eksperymentu

	TML_MTR_INST[i]._cfg.maxVel = 8000.0/60.0/TML_MTR_INST[i]._cfg.rev_motor/ TML_MTR_INST[i]._cfg.rev_scale;
	TML_MTR_INST[i]._cfg.maxAcc = TML_MTR_INST[i]._cfg.maxVel * 10.0 ;
	TML_MTR_INST[i]._cfg.absLastPos = OLD_MTR_POS[TML_AX_OSC];
	TML_MTR_INST[i]._cfg.pAbsLastPos = &OLD_MTR_POS[i];

	TML_MTR_INST[i]._int.kVolt = 1365.0;

	TML_MTR_INST[i]._cfg.absFbk = 10;

	TML_MTR_INST[i]._cfg.HeartBeat = 0.4;
	//TML_MTR_INST[i]._cfg.PVTPeriod = 0.08;

	strcpy(TML_MTR_INST[i]._cfg.programName , "1821_BPV2_OSC.sw");
	TML_MTR_INST[i].ProgramVersion = ASC2UDINT("1821");

	TML_MTR_INST[i].FirmwareVersion = ASC2UDINT("674C");  //0x674B
	TML_MTR_INST[i]._cfg.NotAutoDownload = 1;

	////////////////////////////////////////
	i = TML_AX_TVL;

	strcpy(TML_MTR_INST[i].Name , "TVL");

	// Corrected 29May19
	//TML_MTR_INST[i]._cfg.loopPeriod = 0.0005; // Slow loop
	TML_MTR_INST[i]._cfg.loopPeriod = 0.001; // Slow loop
	// It was in BPV
	TML_MTR_INST[i]._cfg.units = 1024 * 4; //
	TML_MTR_INST[i]._cfg.rev_motor = 156;
	TML_MTR_INST[i]._cfg.rev_scale = 1.0 /( 1.25 * 25.4 * M_PI) ;

	TML_MTR_INST[i]._cfg.maxVel = fabsf(4500.0/60.0/TML_MTR_INST[i]._cfg.rev_motor/ TML_MTR_INST[i]._cfg.rev_scale);
	TML_MTR_INST[i]._cfg.maxAcc = TML_MTR_INST[i]._cfg.maxVel * 10.0 ;
	TML_MTR_INST[i]._cfg.absLastPos = OLD_MTR_POS[i];
	TML_MTR_INST[i]._cfg.absFbk = 2;

	TML_MTR_INST[i]._cfg.HeartBeat = 0.2;

	strcpy(TML_MTR_INST[i]._cfg.programName , "1625_BPV2_TVL.sw");
	TML_MTR_INST[i].ProgramVersion = ASC2UDINT("1625");

	TML_MTR_INST[i].FirmwareVersion = ASC2UDINT("6A2B");  //0x674B
	TML_MTR_INST[i]._cfg.Appl_ID_adr = 0x7FCF;
	TML_MTR_INST[i]._cfg.NotAutoDownload = 1;

	///////////////////////////////////////////////////
	i = TML_AX_INDX;

	strcpy(TML_MTR_INST[i].Name , "INDX");

	// Analog Feedback from REF
	TML_MTR_INST[i]._cfg.loopPeriod = 0.001;

	TML_MTR_INST[i]._cfg.units = 500 * 4;
	TML_MTR_INST[i]._cfg.rev_motor = 24;
	TML_MTR_INST[i]._cfg.rev_scale = 1.0/5.0;
	TML_MTR_INST[i]._cfg.maxVel = 10000.0; //
	TML_MTR_INST[i]._cfg.maxAcc = 100.0;
	TML_MTR_INST[i]._cfg.absFbk = 0;

	TML_MTR_INST[i]._cfg.HeartBeat = 0.4;

	strcpy(TML_MTR_INST[i]._cfg.programName , "0326_BPV_WP.sw");
	TML_MTR_INST[i].ProgramVersion = ASC2UDINT("0326");

	TML_MTR_INST[i].FirmwareVersion = ASC2UDINT("6A2B");
	TML_MTR_INST[i]._cfg.Appl_ID_adr = 0x7FCF;
	TML_MTR_INST[i]._cfg.NotAutoDownload = 1;

	////////////////////////////////////////////
	i = TML_AX_AHC;

	strcpy(TML_MTR_INST[i].Name , "AHC");

	// Analog Feedback from REF
	TML_MTR_INST[i]._cfg.loopPeriod = 0.001;
	TML_MTR_INST[i]._cfg.units = 4096;
	TML_MTR_INST[i]._cfg.rev_motor = 1;
	TML_MTR_INST[i]._cfg.rev_scale = 1.0/5.0;
	TML_MTR_INST[i]._cfg.maxVel = 1500.0;
	TML_MTR_INST[i]._cfg.maxAcc = TML_MTR_INST[i]._cfg.maxVel * 10.0;
	//TML_MTR_INST[i]._cfg.satpMax = 27853; // KPP bylo Stauration of proportional gain
	TML_MTR_INST[i]._cfg.satpMax = 32000; // KPP bylo Stauration of proportional gain
	//TML_MTR_INST[i]._cfg.kppMax = 32000; // KPP bylo Stauration of proportional gain
	//TML_MTR_INST[i]._cfg.kipMax = 200; // KPP bylo Stauration of proportional gain
	TML_MTR_INST[i]._cfg.kppMax = 32000;
	TML_MTR_INST[i]._cfg.kipMax = 1000;
	TML_MTR_INST[i]._cfg.absFbk = 0;

	TML_MTR_INST[i]._cfg.HeartBeat = 0.8;

	//TML_MTR_INST[i]._cfg.signFilter = curCfg->Param[parAVC_FbkFilter].val[0];

	strcpy(TML_MTR_INST[i]._cfg.programName , "1526_SMH_AVC.sw");
	TML_MTR_INST[i].ProgramVersion = ASC2UDINT("1526");

	TML_MTR_INST[i].FirmwareVersion = ASC2UDINT("6A2B");  //0x674C , 514D
	TML_MTR_INST[i]._cfg.Appl_ID_adr = 0x7FCF;
	TML_MTR_INST[i]._cfg.NotAutoDownload = 1;

	//TML_MTR_INST[i]._cfg.sftLimitPos = 0.0;
	//TML_MTR_INST[i]._cfg.sftLimitNeg = 0.0;

	TML_MTR_INST[i]._cfg.AnalLimitPos = 3900;
	TML_MTR_INST[i]._cfg.AnalLimitNeg = 100;

	TML_MTR_INST[i]._cfg.MtrType = 1 ; // 3phase brusshless

	////////////////////////////////////////////
	i = TML_AX_WF;
	strcpy(TML_MTR_INST[i].Name , "WF");

	// Analog Feedback from REF
	TML_MTR_INST[i]._cfg.loopPeriod = 0.001;
	TML_MTR_INST[i]._cfg.units = 1024 * 4; //

	TML_MTR_INST[i]._cfg.rev_scale = 1.0 /( 0.75 * 25.4 * M_PI) ;
	TML_MTR_INST[i]._cfg.rev_motor = 35.0;

	TML_MTR_INST[i]._cfg.maxVel = 520 * 25.4/ 60.0; //// 520 ipm
	TML_MTR_INST[i]._cfg.maxAcc = TML_MTR_INST[i]._cfg.maxVel * 4.0;
	TML_MTR_INST[i]._cfg.absFbk = 0;

	TML_MTR_INST[i]._cfg.HeartBeat = 0.4;

	strcpy(TML_MTR_INST[i]._cfg.programName , "0325_BPV_WF.sw");
	TML_MTR_INST[i].ProgramVersion = ASC2UDINT("0325");

	TML_MTR_INST[i].FirmwareVersion = ASC2UDINT("6A2B");
	TML_MTR_INST[i]._cfg.Appl_ID_adr = 0x7FCF;
	TML_MTR_INST[i]._cfg.NotAutoDownload = 1;

	/***********************************************************/
	/***************************************************************/
	/////////////////////////////////////////////////////////////////

	TML_MTR_INST[TML_AX_TVL].pState = &VectorStateMach[VECT_AX_TVL];
	TML_MTR_INST[TML_AX_OSC].pState = &VectorStateMach[VECT_AX_OSC];
	TML_MTR_INST[TML_AX_INDX].pState = &VectorStateMach[VECT_AX_INDX];
	TML_MTR_INST[TML_AX_AHC].pState = &VectorStateMach[VECT_AX_AHC];
	TML_MTR_INST[TML_AX_WF].pState = &VectorStateMach[VECT_AX_WF];

	strcpy(VectorStateMach[VECT_AX_TVL].Name , TML_MTR_INST[TML_AX_TVL].Name);
	strcpy(VectorStateMach[VECT_AX_OSC].Name , TML_MTR_INST[TML_AX_OSC].Name);
	strcpy(VectorStateMach[VECT_AX_INDX].Name , TML_MTR_INST[TML_AX_INDX].Name);
	strcpy(VectorStateMach[VECT_AX_AHC].Name , TML_MTR_INST[TML_AX_AHC].Name);
	strcpy(VectorStateMach[VECT_AX_WF].Name , TML_MTR_INST[TML_AX_WF].Name);

	TML_mgr[0].hrdw[0].AxisNum = 0;
	TML_mgr[0].hrdw[1].AxisNum = 5;

	TML_mgr[0].pAxis[0] = 0;
	TML_mgr[0].pAxis[1] = &AxisCh[0];

	TML_mgr[0].pTML[0] = 0;
	TML_mgr[0].pTML[1] = &TML_MTR_INST[0];

	AxisCh[TML_AX_TVL].AxisID	= 25;	// BPV2 - TVL
	AxisCh[TML_AX_OSC].AxisID 	= 21;	// BPV2 - OSC
	AxisCh[TML_AX_INDX].AxisID 	= 6;	// BPV2 - WP
	AxisCh[TML_AX_AHC].AxisID 	= 26; 	// BPV2 - AVC
	AxisCh[TML_AX_WF].AxisID 	= 5;	// BPV2 - WF

	/// Tak jest w BPV2

	/*
	AxisCh[TML_AX_TVL].AxisID	= 25;
	AxisCh[TML_AX_OSC].AxisID 	= 21;
	AxisCh[TML_AX_AVC].AxisID 	= 26;
	AxisCh[TML_AX_WRST].AxisID 	= 23;

	AxisCh[TML_AX_INDX].AxisID 	= 22;
	AxisCh[TML_AX_INDX_1].AxisID 	= 24;

	AxisCh[TML_AX_WF].AxisID 	= 5;
	AxisCh[TML_AX_WP].AxisID 	= 6;
	AxisCh[TML_AX_WF_1].AxisID 	= 7;
	AxisCh[TML_AX_WP_1].AxisID 	= 8;
	*/

}
#endif
void _CYCLIC ProgramCyclic(void)
{int i , k ;

	LoggerSrv(&LogMgr);

/*
	if(ErrorMgr.Error){

		k = ErrorMgr.lastItemIndx - 5;
		if( k < 0)
			k =0;

		for(i = 0 ; i < 5 ; i++){

			if((k + i)<= ErrorMgr.lastItemIndx){

				if((ErrorMgr.history[k + i]>=ERROR_DRV_01)
					&& (ErrorMgr.history[k + i] < ERROR_DRV_41)){

					AssignMtrErrorText(ErrorMgr_Txt[i] , ErrorMgr.history[k + i] , ErrorMgr.logs[ErrorMgr.history[k + i]].value);

				}
				else
					xsprintf(ErrorMgr_Txt[i], "%s: %X" , ErrorMgr.logs[ErrorMgr.history[k + i]].txt , ErrorMgr.logs[ErrorMgr.history[k + i]].value);
			}
			else
				strcpy(ErrorMgr_Txt[i] , " -------------- ");

		}
	}
*/
}

void _EXIT ProgramExit(void)
{

}

void AssignMtrErrorText(char* txt , UDINT i , UDINT val ){

plcstring errortxt[64];

	if(i < ERROR_DRV_11)
		xsprintf(txt, "Drive: %s: " , TML_MTR_INST[i-1].Name);
	else if(i < ERROR_DRV_21)
		xsprintf(txt, "Drive: %s: " , TML_MTR_INST[i - ERROR_DRV_11].Name);
	else if(i < ERROR_DRV_31)
		xsprintf(txt, "Drive: %s: " , TML_MTR_INST[i- ERROR_DRV_21].Name);
	else if(i < ERROR_DRV_41)
		xsprintf(txt, "Drive: %s: " , TML_MTR_INST[i- ERROR_DRV_31].Name);

	switch(val){

		case 1: strcat(txt , "CANbus Error"); 			break;

		case 2: strcat(txt , "Short-Circuit Error"); 		break;

		case 3: strcat(txt , "Invalid Setup Error"); 		break;

		case 4: strcat(txt , "Control (Position) Error "); 		break;

		case 5: strcat(txt , "Serial Comm Error"); 		break;

		case 6: strcat(txt , "Feedback Error"); 		break;

		case 7: strcat(txt , "POT Limit Error"); 			break;

		case 8: strcat(txt , "NOT Limit Error"); 			break;

		case 9: strcat(txt , "Instantanious Over-Current Error"); 			break;

		case 10: strcat(txt , "I2t Over-Current Error"); 					break;

		case 11: strcat(txt , "Over-Temperature Error - Motor"); 	break;

		case 12: strcat(txt , "Over-Temperature Error - Drive"); 	break;

		case 13: strcat(txt , "Over-Voltage Error"); 		break;

		case 14: strcat(txt , "Under-Voltage Error"); 		break;

		case 15: strcat(txt , "Command Error"); 		break;

		case 16: strcat(txt , "E-Stop Enable Inactive Error"); 	break;

		case 17: strcat(txt , "Init Error"); 	break;

		case 18: strcat(txt , "No Comunnication"); 	break;

		default: xsprintf(txt+strlen(txt), "Unknown Error %X " , val);

	}

}
```

### Program Logical/MainProc (ANSIC)
